{attribute 'linkalways'} 
{attribute 'no_explicit_call' := 'This FB is a CLASS and must be accessed using methods or properties'}
{attribute 'enable_dynamic_creation'}
FUNCTION_BLOCK _ETcVnDrawShape EXTENDS EnumDatatypeBase
VAR
	localData : ETcVnDrawShape;
	activeData : REFERENCE TO ETcVnDrawShape;
	enumBaseDatatype : _DINT(localData);
END_VAR

METHOD PRIVATE AddLocalEnumeration
VAR_INPUT
	Enumeration : T_MAXSTRING;
	Value : ETcVnDrawShape;
END_VAR
AddEnumeration(Enumeration, Value);
END_METHOD

PROPERTY PUBLIC Address : PVOID
GET
Address := ADR(activeData);
END_GET
END_PROPERTY

METHOD PUBLIC ClearReference
VAR_INPUT
END_VAR
activeData REF= localData;
SetBaseDatatypeReference();
END_METHOD

METHOD PUBLIC Clone : I_Datatype
VAR
    pClone : POINTER TO _ETcVnDrawShape;
END_VAR
pClone := __NEW(_ETcVnDrawShape(InitialValue := Value));
Clone := pClone^;
END_METHOD

METHOD FB_init : BOOL
VAR_INPUT
	bInitRetains : BOOL; // if TRUE, the retain variables are initialized (warm start / cold start)
	bInCopyCode : BOOL;  // if TRUE, the instance afterwards gets moved into the copy code (online change)
	InitialValue : ETcVnDrawShape;
END_VAR
localData := InitialValue;
AddBaseDatatype(enumBaseDatatype);
ClearReference();

AddLocalEnumeration('TCVN_DS_RANDOM', ETcVnDrawShape.TCVN_DS_RANDOM);
AddLocalEnumeration('TCVN_DS_CIRCLE', ETcVnDrawShape.TCVN_DS_CIRCLE);
AddLocalEnumeration('TCVN_DS_SQUARE', ETcVnDrawShape.TCVN_DS_SQUARE);
AddLocalEnumeration('TCVN_DS_PLUS', ETcVnDrawShape.TCVN_DS_PLUS);
AddLocalEnumeration('TCVN_DS_X', ETcVnDrawShape.TCVN_DS_X);
AddLocalEnumeration('TCVN_DS_DIAMOND', ETcVnDrawShape.TCVN_DS_DIAMOND);
AddLocalEnumeration('TCVN_DS_MAX', ETcVnDrawShape.TCVN_DS_MAX);
END_METHOD

PROPERTY PUBLIC Identifier : T_MAXSTRING
GET
Identifier := 'ETcVnDrawShape';
END_GET
END_PROPERTY

METHOD IsEnumeratorValueEqual : BOOL
VAR_INPUT
	Enumerator : I_KeyValueForwardEnumerator;
END_VAR
VAR
	storedValue : ETcVnDrawShape;
END_VAR
IF NOT Enumerator.TryGet(storedValue) THEN
	RETURN;
END_IF

IsEnumeratorValueEqual := storedValue = activeData;
END_METHOD

METHOD PUBLIC MakeReferenceTo
VAR_INPUT
	ReferenceTarget : REFERENCE TO ETcVnDrawShape;
END_VAR
activeData REF= ReferenceTarget;
SetBaseDatatypeReference();
END_METHOD

METHOD PROTECTED SetBaseDatatypeReference
VAR_INPUT
END_VAR
enumBaseDatatype.MakeReferenceTo(activeData);
END_METHOD

PROPERTY PUBLIC Size : UDINT
GET
Size := SIZEOF(activeData);
END_GET
END_PROPERTY

METHOD TryMakeReferenceTo : BOOL
VAR_INPUT
	Target : I_Datatype;
END_VAR
VAR
	targetAsEnum : I_EnumDatatype;
	pTargetData : POINTER TO ETcVnDrawShape;
END_VAR
IF NOT Target.TryResolveAsEnumDatatype(targetAsEnum) THEN
	RETURN;
END_IF

IF targetAsEnum.Identifier <> Identifier THEN
	RETURN;
END_IF

pTargetData := Target.Address;
activeData REF= pTargetData^;
SetBaseDatatypeReference();
TryMakeReferenceTo := TRUE;
END_METHOD

PROPERTY PUBLIC Value : ETcVnDrawShape
GET
Value := activeData;
END_GET
SET
activeData := Value;
END_SET
END_PROPERTY

END_FUNCTION_BLOCK

(* stored: Version 1.1.0.1
   POU _ETcVnDrawShape: Id {99f22db0-c968-455e-9096-07a1c6aee15c}, SpecialFunc None
   Folder Constructor: Id {ccf63e7c-5d8a-4b24-a01c-e2dd34eee327}
   Folder Private: Id {e75dda3b-8c08-447e-a138-b518e2414782}
   Folder Protected: Id {84e3bfcb-96b2-4b11-afa2-82a7b4dd128e}
   Method AddLocalEnumeration: Id {4f7948c1-0784-4125-b4a1-56daace4025f}
   Property Address: Id {db320fb1-34a7-4d76-931f-90847ae6664b}
   Get Get: Id {d2322e8a-740c-4b57-af32-b4eff86bc7cd}
   Method ClearReference: Id {7e561e28-0834-447a-b5a2-a7a9c7e8c283}
   Method Clone: Id {15fd3978-34a9-4564-88fa-408526e8852f}
   Method FB_init: Id {2b06fc22-f858-45f4-bcac-19507d194173}
   Property Identifier: Id {7ab40637-a3da-4e65-8a52-87b9779d49e3}
   Get Get: Id {5851186b-29e3-4afc-8da7-98eff0db43f0}
   Method IsEnumeratorValueEqual: Id {a9c52f8d-c600-484b-abca-4630cc7b28da}
   Method MakeReferenceTo: Id {0a625299-18bf-4ca4-8dda-30d49cb44c70}
   Method SetBaseDatatypeReference: Id {95916bf3-f385-474b-abe1-220638c0f566}
   Property Size: Id {b1080d62-bef2-40d2-8567-a210cf5597b2}
   Get Get: Id {f40c17b7-0d4b-435f-8283-fb618d7f4aba}
   Method TryMakeReferenceTo: Id {c6ad6e5e-fd96-4235-9b42-174e44b042d1}
   Property Value: Id {0820feda-1bae-4bf5-ab3e-f3b7413acae1}
   Get Get: Id {f751679e-aeb7-4663-9f7e-a0da631bd845}
   Set Set: Id {f84b1239-3270-4c38-8656-622d748a6637} *)
